{attribute addProperty BoxType "EL2911-0000-0016"}
{attribute addProperty Id "FSOEAT %I*FSOE_09814BC5486"}
{attribute addProperty CRC "486959772"}
{attribute addProperty SizeInBites "48"}
{attribute addProperty SizeInBytes "6"}
TYPE FSoE_Inputs_1D066A9C :
STRUCT
	{attribute addProperty Name "FSOE"}
	FSOE AT %I* : FSOE_09814BC5;
END_STRUCT
END_TYPE

(* stored: Version 1.2.0.0, ProductVersion 3.1.4024.9
   DUT FSoE_Inputs_1D066A9C: Id {59fdc867-f05d-4883-a118-dcdf9fd24064} *)
